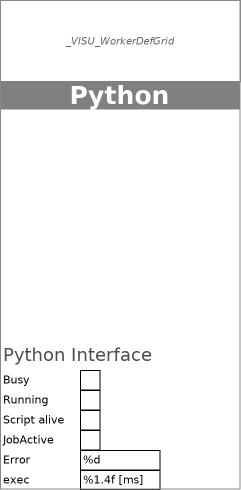
VISUALIZATION _VISU_WorkerDefGrid_Python  // 241x490
VAR_IN_OUT
		m_Inst : FB_WorkerDefGrid_Python;
END_VAR
    Frame (0,0 241x82)
        shows _VISU_WorkerDefGrid(m_Inst := m_Inst)
    Label (0,340 240x30), "Python Interface"
    Rectangle (80,450 80x20), "%d", text variable: m_Inst.fbPythonInterface.nErrorId, colour toggle: m_Inst.fbPythonInterface.bError
        tap m_Inst.fbPythonInterface._bResetError
    Rectangle (0,450 40x20), "Error"
    Rectangle (80,470 80x20), "%1.4f [ms]", text variable: m_Inst.fbPythonInterface.tWatchdogTime
    Rectangle (0,470 40x20), "exec"
    Rectangle (0,80 240x30), "Python", colour toggle: m_Inst._pAttachedCt <> 0
    Rectangle (0,370 80x20), "Busy"
    RoundedRectangle (80,370 20x20), colour toggle: m_Inst.fbPythonInterface.bBusy
    Rectangle (0,390 80x20), "Running"
    RoundedRectangle (80,390 20x20), colour toggle: m_Inst.fbPythonInterface.bRunning
    Rectangle (0,430 80x20), "JobActive"
    RoundedRectangle (80,430 20x20), colour toggle: m_Inst.fbPythonInterface.bJobActive
    Rectangle (0,410 80x20), "Script alive"
    RoundedRectangle (80,410 20x20), colour toggle: m_Inst.fbPythonInterface.bScriptAlive
END_VISUALIZATION

(* stored: Version 1.1.0.1, ProductVersion 3.1.4024.3
   Visu _VISU_WorkerDefGrid_Python: Id {792c7fd0-0dda-4fa8-9735-c805c7cc0638} *)
